PROGRAM MAIN
VAR
	INMODE : INMODE;
	
	Timer : TON;
	TimerT : TIME;
	TimerSW : BOOL;
	
	FallTrig : F_TRIG;
	FallTrigCLK : BOOL;
	
	RiseTrig : R_TRIG;
	RiseTrigCLK : BOOL;
	
	Pulse : Pulse;
	PulseSIGNAL : BOOL; 
	PulseTime : TIME;
	
	N1: INT;
	N2: INT;
	Task : WSTRING;
	Task2: WSTRING;
	Logs : WSTRING;
	
	Carry_IN : BOOL;
	Press : BOOL;
	Track_IN : BOOL;
	Alert_1 : BOOL;
	LiftUP : BOOL;
	Lift_DOWN : BOOL;
	Lift_END : BOOL;
	Lift_IN  : BOOL;
	Palett_IN : BOOL;
	Palett_GRAB : BOOL;
	Palett_PUSH : BOOL;
	Flap : BOOL;
	Palett_OPEN : BOOL;
	Track_OUT : BOOL;
	Horn : BOOL;
	Alert_2 : BOOL;
	
	Carry_IN_FULL : BOOL;
	Press_FULL : BOOL;
	Press_END : BOOL;
	System_OK : BOOL;
	Track_IN_EMPTY : BOOL;
	Track_OUT_EMPTY : BOOL;
	Lift_FRONT : BOOL;
	Lift_BACK : BOOL;
	Lift_RUN : BOOL;
	Palett_PUSH_END : BOOL;
	Palett_CLOSED : BOOL;
	Palett_GRAB_OK : BOOL;
	Auto_SWITCH : BOOL;
	START : BOOL;
	STOP : BOOL;
	RESET : BOOL;
	
	BOX_Count : INT := 0;
	Line_Count : INT := 0;
	Layer_Count : INT := 0;
	RAK_Count : INT := 0;
	
	Stack_MODE : BOOL := TRUE; //if 1 then 3x2; if 0 then 2x3
	Layer_READY : BOOL;
	
	BOX_Count_FULL : BOOL;
	Line_Count_FULL : BOOL;
	
END_VAR

INMODE(); 

Timer(IN:=TimerSW,PT:=TimerT);
FallTrig(CLK:=FallTrigCLK);
RiseTrig(CLK:=Carry_IN_FULL);
Pulse(SIGNAL:=PulseSIGNAL,Pulse_time:=PulseTime);

GIOL.TaskName := Task;
GIOL.CaseNum := N1;

GIOL.TaskName2 := Task2;
GIOL.CaseNum2 := N2;

Carry_IN_FULL := GIOL.In0;
Press_FULL := GIOL.In1;
Press_END := GIOL.In3;
System_OK := GIOL.In2;
Track_IN_EMPTY := GIOL.In4;
Track_OUT_EMPTY := GIOL.In7;
Lift_FRONT := GIOL.In5;
Lift_BACK := GIOL.In6;
Lift_RUN := GIOL.In8;
Palett_PUSH_END := GIOL.In9;
Palett_CLOSED := GIOL.In10;
Palett_GRAB_OK := GIOL.In11;
Auto_SWITCH := GIOL.In12;
START := GIOL.In13;
STOP := GIOL.In14;
RESET := GIOL.In15;

GIOL.Out0 := Carry_IN;
GIOL.Out1 := Press;
GIOL.Out2 := Track_IN;
GIOL.Out3 := Alert_1;
GIOL.Out4 := LiftUP;
GIOL.Out5 := Lift_DOWN;
GIOL.Out6 := Lift_END;
GIOL.Out7 := Lift_IN;
GIOL.Out8 := Palett_PUSH;
GIOL.Out9 := Palett_GRAB;
GIOL.Out10 := Palett_IN;
GIOL.Out11 := Flap;
GIOL.Out12 := Palett_OPEN;
GIOL.Out13 := Track_OUT;
GIOL.Out14 := Horn;
GIOL.Out15 := Alert_2;

//STACK MODE
IF Stack_MODE THEN
	Flap:=FALSE;
	IF Line_Count = 3 THEN
			Line_Count := 0;
			Line_Count_FULL :=TRUE;
			Layer_Count := Layer_Count +1;
	END_IF
	IF BOX_Count = 3 THEN
		BOX_Count := 1;
		BOX_Count_FULL := TRUE;
	END_IF
ELSE
	Flap:=TRUE;
	IF Line_Count = 2 THEN
			Line_Count := 0;
			Line_Count_FULL :=TRUE;
			Layer_Count := Layer_Count +1;
	END_IF
	IF BOX_Count = 4 THEN
		BOX_Count := 0;
		BOX_Count_FULL := TRUE;
	END_IF
	
END_IF

IF Layer_Count = 3 THEN
	Layer_Count := 0;
	Stack_MODE  := NOT Stack_MODE;
END_IF

// PRESS {
IF Press THEN
	Press:=FALSE;
END_IF

IF Press_FULL AND Press_END THEN
	Press:=TRUE;
END_IF
//} Press

IF RiseTrig.Q THEN
	BOX_Count := BOX_Count + 1;
END_IF

//Async TASK_1 { Carry_IN, Palett_ALL
//
CASE N1 OF
	
	0:Task:="Building first line";
		Carry_IN := TRUE;
		Palett_IN := TRUE;
		Palett_OPEN := FALSE;
		N1:=10;
		
	10:Task:="Building first line";	
		IF BOX_Count_FULL THEN
			Carry_IN := FALSE;
			Palett_IN := FALSE;
			Palett_PUSH := TRUE;
			BOX_Count :=1;
			TimerT:=T#3500MS;
			BOX_Count_FULL := FALSE;
			N1:=20;
		END_IF
		
	20:Task:="Stop Boxes and push line";
		TimerSW:=TRUE;
		IF Timer.Q THEN
			Line_Count := Line_Count + 1;
			TimerSW := FALSE;
			Palett_PUSH := FALSE;
			N1:=30;
		END_IF
		
	30:Task:="Stop Boxes and push line";
		TimerSW := TRUE;
		IF Timer.Q THEN
			TimerSW:=FALSE;
			N1:= 0;
		END_IF
		IF Line_Count_FULL THEN
			N1:=60;
			Line_Count_FULL := FALSE;
			Palett_GRAB := TRUE;
		END_IF
		
	60:Task:="";
		IF Palett_GRAB_OK THEN
			Palett_OPEN:=TRUE;
			TimerT:=T#3S;
			N1:=70;
		END_IF
		
	70:Task:="";
		TimerSW:=TRUE;
		IF Timer.Q THEN
			Palett_GRAB := FALSE;
			TimerSW:=FALSE;
			N1:=0;
		END_IF
	ELSE
		N1:=0;
END_CASE
//} Async TASK_1

//Async TASK_2 { Rack, 
CASE N2 OF
	0:Task2:="";
	ELSE
		N2:=0;
END_CASE
//} Async TASK_2

END_PROGRAM

(* stored: Version 1.1.0.1, ProductVersion 3.1.4024.15
   POU MAIN: Id {55f2dad4-fae0-4be3-a7be-b728afd4fa9e}, SpecialFunc None *)
